ABB RobotStudio station: ProyectoC1.rspag

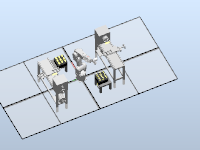
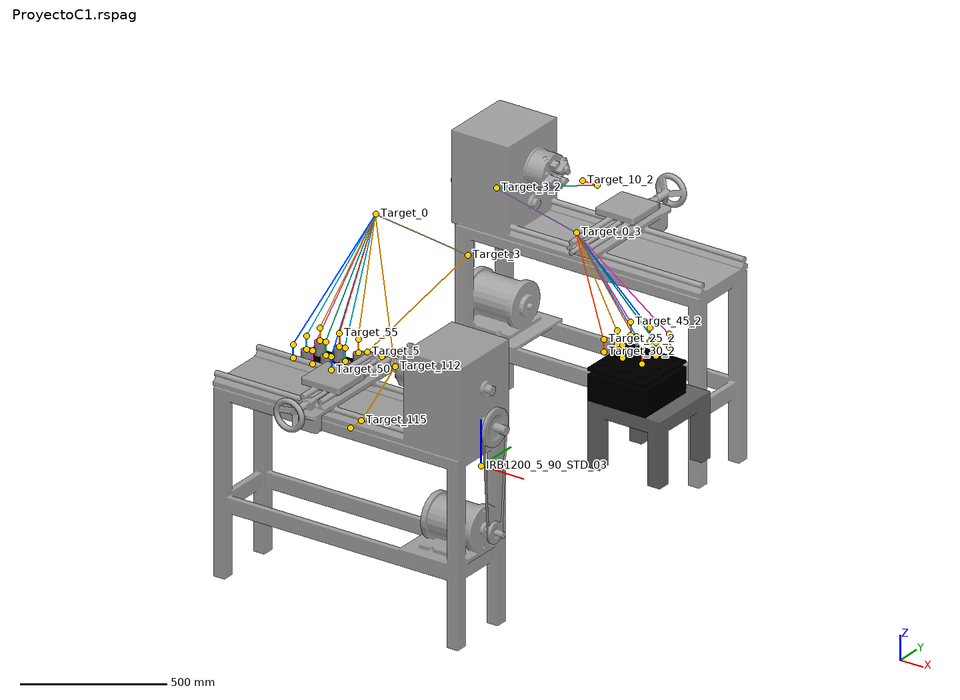
[picture v1: parts stored in the station drawn from their meshes, with robot base, taught points and paths (robot models come from the ABB library and are not in the file)]
--- station ---
Station Prueba1 (saved by RobotStudio 21.2.9526.0)
Controller Controller8
  mechanical unit ROB_1: IRB1200_5_90_STD_03, 6 joints, base frame (0, 0, 0) mm, rotated rx 0 ry 0 rz 180 deg
Layout (positions relative to the parent item):
  - Part_10 [part] at (300, 200, 0) mm, size 304.8 x 304.8 x 257.1 mm
  - IRB1200_5_90_STD_03 [mechanism, from Robots\IRB1200_5_90_STD_03.rslib] at (0, 0, 0) mm, rotated rx 0 ry 0 rz 180 deg; joint values [0.2272, -0.2553, -0.0183, 1.0645, 1.1707, 0.1682] (rad or m)
  - Pieza mecanizada_2 [part] at (-340.99, -320.29, 378.02) mm, rotated rx 0.01 ry 0 rz -1.08 deg, size 40.5 x 40.5 x 50.8 mm
  - Pieza mecanizada_3 [part] at (-340.26, -399.91, 378.02) mm, rotated rx 0 ry 0 rz 0.16 deg, size 40.5 x 40.5 x 50.8 mm
  - Pieza mecanizada_4 [part] at (-420.52, -241.71, 378.02) mm, rotated rx 0 ry 0 rz 2.15 deg, size 40.5 x 40.5 x 50.8 mm
  - Pieza mecanizada_5 [part] at (-420.06, -320.35, 378.02) mm, rotated rx 0 ry 0 rz 0.63 deg, size 40.5 x 40.5 x 50.8 mm
  - Pieza mecanizada_6 [part] at (-419.99, -400.08, 378.02) mm, size 40.5 x 40.5 x 50.8 mm
  - Pieza mecanizada_7 [part] at (-500.46, -240.05, 378.02) mm, rotated rx 0 ry 0 rz 0.98 deg, size 40.5 x 40.5 x 50.8 mm
  - Pieza mecanizada_8 [part] at (-500, -320, 378.02) mm, rotated rx 0 ry 0 rz 0.01 deg, size 40.5 x 40.5 x 50.8 mm
  - Pieza mecanizada_9 [part] at (-500, -400, 378.02) mm, rotated rx 0 ry 0 rz 0.01 deg, size 40.5 x 40.5 x 50.8 mm
  - Gripper_triple [mechanism] at (-326.49, -143.26, 968.24) mm, rotated rx 109.8 ry 16.48 rz -12.76 deg
      TCP Tool_acople at (0, -72.83, 94.3) mm, rotated rx 45 ry 0 rz 0 deg
      TCP Tool_desacople at (-1.73, 75.04, 92.27) mm, rotated rx -45 ry 0 rz 0 deg
      TCP Refrigerator at (40, 0, 44) mm, rotated rx 0 ry 90 rz 0 deg
      links: Herramienta
  - Torno_1 [smart component]
      signals: DO Finish, DO Mounted, DI Start, DI Attach, DI Detach
      connections:
        Torno_1.Start -> Timer_2.Active
        Timer_2.Output -> Torno_1.Finish
        Torno_1.Start -> LogicGate.InputA
        LogicGate.Output -> Detacher_10.Execute
        LineSensor.SensorOut -> Torno_1.Mounted
        Torno_1.Start -> Attacher.Execute
        LogicGate.Output -> Attacher_12.Execute
        Torno_1.Start -> Detacher_12.Execute
        LineSensor.SensedPart => Attacher.Child
        LineSensor.SensedPart => Detacher_10.Child
        LineSensor.SensedPart => Attacher_12.Child
        LineSensor.SensedPart => Detacher_12.Child
    - Torno [part] at (-288, 524, 0) mm, size 1289.1 x 1431.5 x 1343.8 mm
    - Detacher_10 [smart component, from Components\Detacher.rslib]
        properties: Child=Pieza mecanizada; KeepPosition=true
    - Attacher [smart component, from Components\Attacher.rslib]
        properties: Parent=Torno; Flange=0; Child=Pieza mecanizada; Mount=false; Offset=[0 0 0]; Orientation=[0 0 0]
    - LogicGate [smart component, from Components\LogicGate.rslib]
        properties: Operator=NOT; Delay=0
    - LineSensor [smart component, from Components\LineSensor.rslib]
        properties: Start=[0.14 -0.8 0.75]; End=[0.14 -0.69 0.75]; Radius=0; SensedPart=Pieza mecanizada; SensedPoint=[0.14 -0.777924682617188 0.75]
      - _sensorPart_ [part], size 0 x 110 x 0 mm
    - Attacher_12 [smart component, from Components\Attacher.rslib]
        properties: Parent=Gripper_triple; Flange=1; Child=Pieza mecanizada; Mount=false; Offset=[0 0 0]; Orientation=[0 0 0]
    - Detacher_12 [smart component, from Components\Detacher.rslib]
        properties: Child=Pieza mecanizada; KeepPosition=true
    - Torno_abierto [part] at (726.53, 140.46, 2.16) mm, size 1118.3 x 604.1 x 1068.7 mm
  - Torno_2 [smart component]
      signals: DO Finish, DO Mounted, DI Start, DI Attach, DI Detach
      connections:
        Torno_2.Start -> Attacher.Execute
        Torno_2.Start -> LogicGate_14.InputA
        LogicGate_14.Output -> Detacher.Execute
        LogicGate_14.Output -> Attacher_2.Execute
        Torno_2.Start -> Detacher_2.Execute
        LineSensor.SensorOut -> Torno_2.Mounted
        LineSensor.SensedPart => Detacher.Child
        LineSensor.SensedPart => Detacher_2.Child
        LineSensor.SensedPart => Attacher_2.Child
        LineSensor.SensedPart => Attacher.Child
    - Torno_3 [part] at (288, -524, 0) mm, rotated rx 0 ry 0 rz 180 deg, size 1289.1 x 1431.5 x 1343.8 mm
    - Attacher [smart component, from Components\Attacher.rslib]
        properties: Parent=Torno_3; Flange=0; Child=(none); Mount=false; Offset=[0 0 0]; Orientation=[0 0 0]
    - Attacher_2 [smart component, from Components\Attacher.rslib]
        properties: Parent=Gripper_triple; Flange=1; Child=(none); Mount=false; Offset=[0 0 0]; Orientation=[0 0 0]
    - Detacher [smart component, from Components\Detacher.rslib]
        properties: Child=(none); KeepPosition=true
    - Detacher_2 [smart component, from Components\Detacher.rslib]
        properties: Child=(none); KeepPosition=true
    - LineSensor [smart component, from Components\LineSensor.rslib]
        properties: Start=[-0.14 0.8 0.75]; End=[-0.14 0.69 0.75]; Radius=0; SensedPart=(none); SensedPoint=[0 0 0]
      - _sensorPart_ [part], size 0 x 110 x 0 mm
    - LogicGate_14 [smart component, from Components\LogicGate.rslib]
        properties: Operator=NOT; Delay=0
    - Torno_abierto_2 [part] at (-725.71, -155.46, 2.16) mm, rotated rx 0 ry 0 rz 180 deg, size 1118.3 x 604.1 x 1068.7 mm
  - Rotador [smart component]
      signals: DI Start, DO Finish, DI Attach, DI Detach
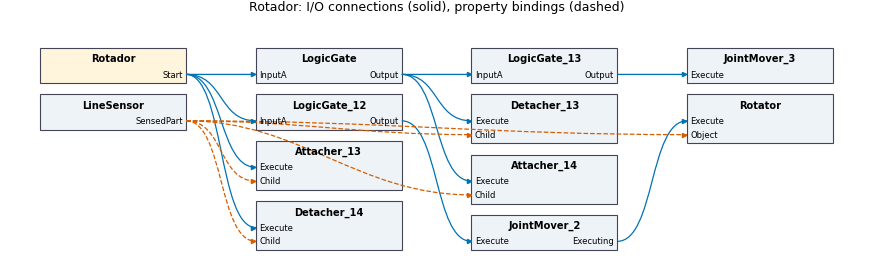
      connections:
        Rotador.Start -> LogicGate.InputA
        Rotador.Start -> Attacher_13.Execute
        LogicGate.Output -> Detacher_13.Execute
        Rotador.Start -> LogicGate_12.InputA
        LogicGate_12.Output -> JointMover_2.Execute
        LogicGate.Output -> Attacher_14.Execute
        Rotador.Start -> Detacher_14.Execute
        JointMover_2.Executing -> Rotator.Execute
        LogicGate.Output -> LogicGate_13.InputA
        LogicGate_13.Output -> JointMover_3.Execute
        LineSensor.SensedPart => Attacher_13.Child
        LineSensor.SensedPart => Detacher_13.Child
        LineSensor.SensedPart => Detacher_14.Child
        LineSensor.SensedPart => Attacher_14.Child
        LineSensor.SensedPart => Rotator.Object
    - My_Mechanism [mechanism] at (0, 0, 0) mm; joint values [0] (rad or m)
        links: L0, L1
    - JointMover_2 [smart component, from Components\JointMover.rslib]
        properties: Mechanism=My_Mechanism; Relative=false; Duration=0.5; J1=3.14159265358979
    - JointMover_3 [smart component, from Components\JointMover.rslib]
        properties: Mechanism=My_Mechanism; Relative=false; Duration=1; J1=0
    - LogicGate [smart component, from Components\LogicGate.rslib]
        properties: Operator=NOT; Delay=0
    - Attacher_13 [smart component, from Components\Attacher.rslib]
        properties: Parent=My_Mechanism; Flange=0; Child=(none); Mount=false; Offset=[0 0 0]; Orientation=[0 0 0]
    - LineSensor [smart component, from Components\LineSensor.rslib]
        properties: Start=[-0.42 -0.225 0.16]; End=[-0.42 -0.225 0.06]; Radius=0; SensedPart=(none); SensedPoint=[0 0 0]
      - _sensorPart_ [part], size 0 x 0 x 100 mm
    - Detacher_13 [smart component, from Components\Detacher.rslib]
        properties: Child=(none); KeepPosition=true
    - LogicGate_12 [smart component, from Components\LogicGate.rslib]
        properties: Operator=OR; Delay=2
    - Attacher_14 [smart component, from Components\Attacher.rslib]
        properties: Parent=Gripper_triple; Flange=0; Child=(none); Mount=false; Offset=[0 0 0]; Orientation=[0 0 0]
    - Detacher_14 [smart component, from Components\Detacher.rslib]
        properties: Child=(none); KeepPosition=true
    - Rotator [smart component, from Components\Rotator.rslib]
        properties: Object=(none); CenterPoint=[-0.54 -0.225 0.108]; Axis=[1 0 0]; Speed=11.8682389135614; Reference=Global; ReferenceObject=(none)
    - Timer [smart component, from Components\Timer.rslib]
        properties: StartTime=0; Interval=0; Repeat=true; CurrentTime=1.512
    - LogicGate_13 [smart component, from Components\LogicGate.rslib]
        properties: Operator=OR; Delay=2
  - Sensor_sin_maquinar [smart component]
      signals: DO Sensor_1_activo, DO Sensor_2_activo, DO Sensor_3_activo, DO Sensor_4_activo, DO Sensor_5_activo, DO Sensor_6_activo, DO Sensor_7_activo, DO Sensor_8_activo, DO Sensor_9_activo
      connections:
        LineSensor_4.SensorOut -> Sensor_sin_maquinar.Sensor_4_activo
        LineSensor_5.SensorOut -> Sensor_sin_maquinar.Sensor_5_activo
        LineSensor_6.SensorOut -> Sensor_sin_maquinar.Sensor_6_activo
        LineSensor_7.SensorOut -> Sensor_sin_maquinar.Sensor_7_activo
        LineSensor_8.SensorOut -> Sensor_sin_maquinar.Sensor_8_activo
        LineSensor_9.SensorOut -> Sensor_sin_maquinar.Sensor_9_activo
        LineSensor.SensorOut -> Sensor_sin_maquinar.Sensor_1_activo
        LineSensor_2.SensorOut -> Sensor_sin_maquinar.Sensor_2_activo
        LineSensor_3.SensorOut -> Sensor_sin_maquinar.Sensor_3_activo
    - Palet_2 [part] at (-300, -200, 250) mm, rotated rx 0 ry 0 rz 180 deg, size 243.8 x 243.8 x 129.5 mm
    - LineSensor [smart component, from Components\LineSensor.rslib]
        properties: Start=[-0.37 -0.240108 0.4]; End=[-0.31 -0.24 0.4]; Radius=0; SensedPart=(none); SensedPoint=[0 0 0]
      - _sensorPart_ [part], size 60 x 0.1 x 0 mm
    - LineSensor_2 [smart component, from Components\LineSensor.rslib]
        properties: Start=[-0.37 -0.32 0.4]; End=[-0.31 -0.32 0.4]; Radius=0; SensedPart=Pieza mecanizada_2; SensedPoint=[-0.361003173828125 -0.32 0.4]
      - _sensorPart_ [part], size 60 x 0 x 0 mm
    - LineSensor_3 [smart component, from Components\LineSensor.rslib]
        properties: Start=[-0.37 -0.4 0.4]; End=[-0.31 -0.4 0.4]; Radius=0; SensedPart=Pieza mecanizada_3; SensedPoint=[-0.360261657714844 -0.4 0.4]
      - _sensorPart_ [part], size 60 x 0 x 0 mm
    - LineSensor_4 [smart component, from Components\LineSensor.rslib]
        properties: Start=[-0.45 -0.24 0.4]; End=[-0.39 -0.24 0.4]; Radius=0; SensedPart=Pieza mecanizada_4; SensedPoint=[-0.440390747070313 -0.24 0.4]
      - _sensorPart_ [part], size 60 x 0 x 0 mm
    - LineSensor_5 [smart component, from Components\LineSensor.rslib]
        properties: Start=[-0.45 -0.32 0.4]; End=[-0.39 -0.32 0.4]; Radius=0; SensedPart=Pieza mecanizada_5; SensedPoint=[-0.440016571044922 -0.319999969482422 0.4]
      - _sensorPart_ [part], size 60 x 0 x 0 mm
    - LineSensor_6 [smart component, from Components\LineSensor.rslib]
        properties: Start=[-0.45 -0.4 0.4]; End=[-0.39 -0.4 0.4]; Radius=0; SensedPart=Pieza mecanizada_6; SensedPoint=[-0.439984832763672 -0.4 0.4]
      - _sensorPart_ [part], size 60 x 0 x 0 mm
    - LineSensor_7 [smart component, from Components\LineSensor.rslib]
        properties: Start=[-0.53 -0.24 0.4]; End=[-0.47 -0.24 0.4]; Radius=0; SensedPart=Pieza mecanizada_7; SensedPoint=[-0.520428344726563 -0.239999984741211 0.4]
      - _sensorPart_ [part], size 60 x 0 x 0 mm
    - LineSensor_8 [smart component, from Components\LineSensor.rslib]
        properties: Start=[-0.53 -0.32 0.4]; End=[-0.47 -0.32 0.4]; Radius=0; SensedPart=Pieza mecanizada_8; SensedPoint=[-0.520002136230469 -0.319999969482422 0.4]
      - _sensorPart_ [part], size 60 x 0 x 0 mm
    - LineSensor_9 [smart component, from Components\LineSensor.rslib]
        properties: Start=[-0.53 -0.4 0.4]; End=[-0.47 -0.4 0.4]; Radius=0; SensedPart=Pieza mecanizada_9; SensedPoint=[-0.520002685546875 -0.399999969482422 0.4]
      - _sensorPart_ [part], size 60 x 0 x 0 mm
  - Sensor_maquinadas [smart component]
      signals: DO Sensor_1_activo, DO Sensor_2_activo, DO Sensor_3_activo, DO Sensor_4_activo, DO Sensor_5_activo, DO Sensor_6_activo, DO Sensor_7_activo, DO Sensor_8_activo, DO Sensor_9_activo, DI Detach
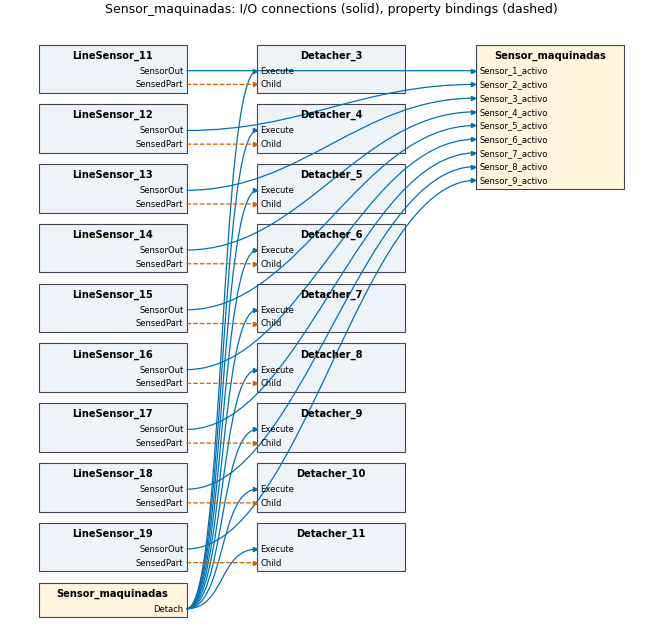
      connections:
        LineSensor_11.SensorOut -> Sensor_maquinadas.Sensor_1_activo
        LineSensor_12.SensorOut -> Sensor_maquinadas.Sensor_2_activo
        LineSensor_13.SensorOut -> Sensor_maquinadas.Sensor_3_activo
        LineSensor_14.SensorOut -> Sensor_maquinadas.Sensor_4_activo
        LineSensor_15.SensorOut -> Sensor_maquinadas.Sensor_5_activo
        LineSensor_16.SensorOut -> Sensor_maquinadas.Sensor_6_activo
        LineSensor_17.SensorOut -> Sensor_maquinadas.Sensor_7_activo
        LineSensor_18.SensorOut -> Sensor_maquinadas.Sensor_8_activo
        LineSensor_19.SensorOut -> Sensor_maquinadas.Sensor_9_activo
        Sensor_maquinadas.Detach -> Detacher_3.Execute
        Sensor_maquinadas.Detach -> Detacher_4.Execute
        Sensor_maquinadas.Detach -> Detacher_5.Execute
        Sensor_maquinadas.Detach -> Detacher_6.Execute
        Sensor_maquinadas.Detach -> Detacher_7.Execute
        Sensor_maquinadas.Detach -> Detacher_8.Execute
        Sensor_maquinadas.Detach -> Detacher_9.Execute
        Sensor_maquinadas.Detach -> Detacher_10.Execute
        Sensor_maquinadas.Detach -> Detacher_11.Execute
        LineSensor_11.SensedPart => Detacher_3.Child
        LineSensor_12.SensedPart => Detacher_4.Child
        LineSensor_13.SensedPart => Detacher_5.Child
        LineSensor_14.SensedPart => Detacher_6.Child
        LineSensor_15.SensedPart => Detacher_7.Child
        LineSensor_16.SensedPart => Detacher_8.Child
        LineSensor_17.SensedPart => Detacher_9.Child
        LineSensor_18.SensedPart => Detacher_10.Child
        LineSensor_19.SensedPart => Detacher_11.Child
    - Palet [part] at (300, 200, 250) mm, size 242.1 x 242.1 x 126.4 mm
    - LineSensor_11 [smart component, from Components\LineSensor.rslib]
        properties: Start=[0.37 0.240108 0.4]; End=[0.31 0.24 0.4]; Radius=0; SensedPart=(none); SensedPoint=[0 0 0]
      - _sensorPart_ [part], size 60 x 0.1 x 0 mm
    - LineSensor_12 [smart component, from Components\LineSensor.rslib]
        properties: Start=[0.37 0.32 0.4]; End=[0.31 0.32 0.4]; Radius=0; SensedPart=Palet; SensedPoint=[0.360499572753906 0.32 0.375]
      - _sensorPart_ [part], size 60 x 0 x 0 mm
    - LineSensor_13 [smart component, from Components\LineSensor.rslib]
        properties: Start=[0.37 0.4 0.4]; End=[0.31 0.4 0.4]; Radius=0; SensedPart=Palet; SensedPoint=[0.360499572753906 0.4 0.375]
      - _sensorPart_ [part], size 60 x 0 x 0 mm
    - LineSensor_14 [smart component, from Components\LineSensor.rslib]
        properties: Start=[0.45 0.24 0.4]; End=[0.39 0.24 0.4]; Radius=0; SensedPart=(none); SensedPoint=[0 0 0]
      - _sensorPart_ [part], size 60 x 0 x 0 mm
    - LineSensor_15 [smart component, from Components\LineSensor.rslib]
        properties: Start=[0.45 0.32 0.4]; End=[0.39 0.32 0.4]; Radius=0; SensedPart=(none); SensedPoint=[0 0 0]
      - _sensorPart_ [part], size 60 x 0 x 0 mm
    - LineSensor_16 [smart component, from Components\LineSensor.rslib]
        properties: Start=[0.45 0.4 0.4]; End=[0.39 0.4 0.4]; Radius=0; SensedPart=(none); SensedPoint=[0 0 0]
      - _sensorPart_ [part], size 60 x 0 x 0 mm
    - LineSensor_17 [smart component, from Components\LineSensor.rslib]
        properties: Start=[0.53 0.24 0.4]; End=[0.47 0.24 0.4]; Radius=0; SensedPart=(none); SensedPoint=[0 0 0]
      - _sensorPart_ [part], size 60 x 0 x 0 mm
    - LineSensor_18 [smart component, from Components\LineSensor.rslib]
        properties: Start=[0.53 0.32 0.4]; End=[0.47 0.32 0.4]; Radius=0; SensedPart=(none); SensedPoint=[0 0 0]
      - _sensorPart_ [part], size 60 x 0 x 0 mm
    - LineSensor_19 [smart component, from Components\LineSensor.rslib]
        properties: Start=[0.53 0.4 0.4]; End=[0.47 0.4 0.4]; Radius=0; SensedPart=(none); SensedPoint=[0 0 0]
      - _sensorPart_ [part], size 60 x 0 x 0 mm
    - Detacher_3 [smart component, from Components\Detacher.rslib]
        properties: Child=(none); KeepPosition=true
    - Detacher_4 [smart component, from Components\Detacher.rslib]
        properties: Child=Palet; KeepPosition=true
    - Detacher_5 [smart component, from Components\Detacher.rslib]
        properties: Child=Palet; KeepPosition=true
    - Detacher_6 [smart component, from Components\Detacher.rslib]
        properties: Child=(none); KeepPosition=true
    - Detacher_7 [smart component, from Components\Detacher.rslib]
        properties: Child=(none); KeepPosition=true
    - Detacher_8 [smart component, from Components\Detacher.rslib]
        properties: Child=(none); KeepPosition=true
    - Detacher_9 [smart component, from Components\Detacher.rslib]
        properties: Child=(none); KeepPosition=true
    - Detacher_10 [smart component, from Components\Detacher.rslib]
        properties: Child=(none); KeepPosition=true
    - Detacher_11 [smart component, from Components\Detacher.rslib]
        properties: Child=(none); KeepPosition=true
  - Attacher [smart component, from Components\Attacher.rslib]
      properties: Parent=Gripper_triple; Flange=0; Child=Pieza mecanizada; Mount=false; Offset=[0 0 0]; Orientation=[0 0 0]
  - Attacher_2 [smart component, from Components\Attacher.rslib]
      properties: Parent=Gripper_triple; Flange=0; Child=Pieza mecanizada_2; Mount=false; Offset=[0 0 0]; Orientation=[0 0 0]
  - Attacher_3 [smart component, from Components\Attacher.rslib]
      properties: Parent=Gripper_triple; Flange=0; Child=Pieza mecanizada_3; Mount=false; Offset=[0 0 0]; Orientation=[0 0 0]
  - Attacher_4 [smart component, from Components\Attacher.rslib]
      properties: Parent=Gripper_triple; Flange=0; Child=Pieza mecanizada_4; Mount=false; Offset=[0 0 0]; Orientation=[0 0 0]
  - Attacher_5 [smart component, from Components\Attacher.rslib]
      properties: Parent=Gripper_triple; Flange=0; Child=Pieza mecanizada_5; Mount=false; Offset=[0 0 0]; Orientation=[0 0 0]
  - Attacher_6 [smart component, from Components\Attacher.rslib]
      properties: Parent=Gripper_triple; Flange=0; Child=Pieza mecanizada_6; Mount=false; Offset=[0 0 0]; Orientation=[0 0 0]
  - Attacher_7 [smart component, from Components\Attacher.rslib]
      properties: Parent=Gripper_triple; Flange=0; Child=Pieza mecanizada_7; Mount=false; Offset=[0 0 0]; Orientation=[0 0 0]
  - Attacher_8 [smart component, from Components\Attacher.rslib]
      properties: Parent=Gripper_triple; Flange=0; Child=Pieza mecanizada_8; Mount=false; Offset=[0 0 0]; Orientation=[0 0 0]
  - Attacher_9 [smart component, from Components\Attacher.rslib]
      properties: Parent=Gripper_triple; Flange=0; Child=Pieza mecanizada_9; Mount=false; Offset=[0 0 0]; Orientation=[0 0 0]
  - Attacher_10 [smart component, from Components\Attacher.rslib]
      properties: Parent=Gripper_triple; Flange=0; Child=(none); Mount=false; Offset=[0 0 0]; Orientation=[0 0 0]
  - LogicGate_2 [smart component, from Components\LogicGate.rslib]
      properties: Operator=AND; Delay=0
  - LogicGate_3 [smart component, from Components\LogicGate.rslib]
      properties: Operator=AND; Delay=0
  - LogicGate_4 [smart component, from Components\LogicGate.rslib]
      properties: Operator=AND; Delay=0
  - LogicGate_5 [smart component, from Components\LogicGate.rslib]
      properties: Operator=AND; Delay=0
  - LogicGate_6 [smart component, from Components\LogicGate.rslib]
      properties: Operator=AND; Delay=0
  - LogicGate_7 [smart component, from Components\LogicGate.rslib]
      properties: Operator=AND; Delay=0
  - LogicGate_8 [smart component, from Components\LogicGate.rslib]
      properties: Operator=AND; Delay=0
  - LogicGate_9 [smart component, from Components\LogicGate.rslib]
      properties: Operator=AND; Delay=0
  - LogicGate_10 [smart component, from Components\LogicGate.rslib]
      properties: Operator=AND; Delay=0
  - Pieza mecanizada [part] at (-339.54, -240.41, 378.02) mm, rotated rx 0 ry 0 rz -1.05 deg, size 40.5 x 40.5 x 50.8 mm
  - Detacher [smart component, from Components\Detacher.rslib]
      properties: Child=Pieza mecanizada; KeepPosition=true
  - Detacher_2 [smart component, from Components\Detacher.rslib]
      properties: Child=Pieza mecanizada_2; KeepPosition=true
  - Detacher_3 [smart component, from Components\Detacher.rslib]
      properties: Child=Pieza mecanizada_3; KeepPosition=true
  - Detacher_4 [smart component, from Components\Detacher.rslib]
      properties: Child=Pieza mecanizada_4; KeepPosition=true
  - Detacher_5 [smart component, from Components\Detacher.rslib]
      properties: Child=Pieza mecanizada_5; KeepPosition=true
  - Detacher_6 [smart component, from Components\Detacher.rslib]
      properties: Child=Pieza mecanizada_6; KeepPosition=true
  - Detacher_7 [smart component, from Components\Detacher.rslib]
      properties: Child=Pieza mecanizada_7; KeepPosition=true
  - Detacher_8 [smart component, from Components\Detacher.rslib]
      properties: Child=Pieza mecanizada_8; KeepPosition=true
  - Detacher_9 [smart component, from Components\Detacher.rslib]
      properties: Child=Pieza mecanizada_9; KeepPosition=true
  - LogicGate_11 [smart component, from Components\LogicGate.rslib]
      properties: Operator=AND; Delay=0
Attachment: Gripper_triple is attached to IRB1200_5_90_STD_03 / Link6
Station signals: DI Execute
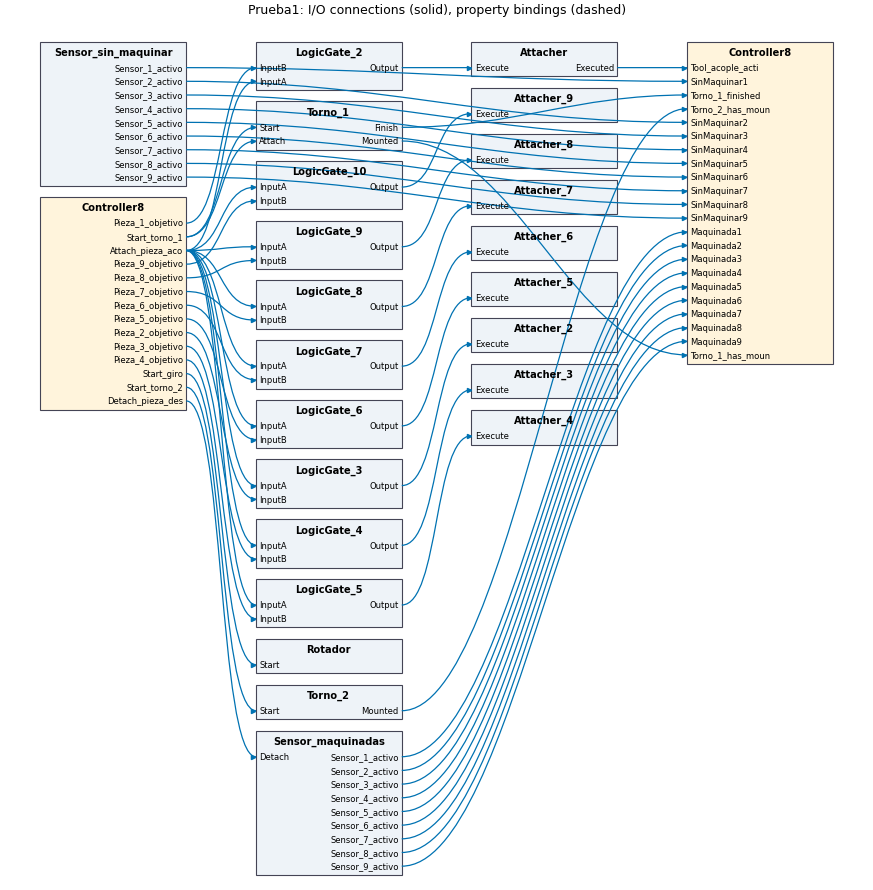
Station logic (signal -> signal, property => property):
  Attacher.Executed -> Controller8.Tool_acople_activa
  Sensor_sin_maquinar.Sensor_1_activo -> Controller8.SinMaquinar1
  Controller8.Pieza_1_objetivo -> LogicGate_2.InputB
  LogicGate_2.Output -> Attacher.Execute
  Controller8.Start_torno_1 -> Torno_1.Start
  Torno_1.Finish -> Controller8.Torno_1_finished
  Controller8.Attach_pieza_acople -> LogicGate_3.InputA
  Controller8.Attach_pieza_acople -> LogicGate_4.InputA
  Controller8.Attach_pieza_acople -> LogicGate_5.InputA
  Controller8.Attach_pieza_acople -> LogicGate_2.InputA
  Controller8.Attach_pieza_acople -> LogicGate_6.InputA
  Controller8.Attach_pieza_acople -> LogicGate_7.InputA
  Controller8.Attach_pieza_acople -> LogicGate_8.InputA
  Controller8.Attach_pieza_acople -> LogicGate_9.InputA
  Controller8.Attach_pieza_acople -> LogicGate_10.InputA
  Controller8.Pieza_9_objetivo -> LogicGate_10.InputB
  Controller8.Pieza_8_objetivo -> LogicGate_9.InputB
  Controller8.Pieza_7_objetivo -> LogicGate_8.InputB
  Controller8.Pieza_6_objetivo -> LogicGate_7.InputB
  Controller8.Pieza_5_objetivo -> LogicGate_6.InputB
  Controller8.Pieza_2_objetivo -> LogicGate_3.InputB
  Controller8.Pieza_3_objetivo -> LogicGate_4.InputB
  Controller8.Pieza_4_objetivo -> LogicGate_5.InputB
  Controller8.Start_torno_1 -> Torno_1.Attach
  Torno_2.Mounted -> Controller8.Torno_2_has_mounted
  Sensor_sin_maquinar.Sensor_2_activo -> Controller8.SinMaquinar2
  Sensor_sin_maquinar.Sensor_3_activo -> Controller8.SinMaquinar3
  Sensor_sin_maquinar.Sensor_4_activo -> Controller8.SinMaquinar4
  Sensor_sin_maquinar.Sensor_5_activo -> Controller8.SinMaquinar5
  Sensor_sin_maquinar.Sensor_6_activo -> Controller8.SinMaquinar6
  Sensor_sin_maquinar.Sensor_7_activo -> Controller8.SinMaquinar7
  Sensor_sin_maquinar.Sensor_8_activo -> Controller8.SinMaquinar8
  Sensor_sin_maquinar.Sensor_9_activo -> Controller8.SinMaquinar9
  LogicGate_3.Output -> Attacher_2.Execute
  LogicGate_4.Output -> Attacher_3.Execute
  LogicGate_5.Output -> Attacher_4.Execute
  LogicGate_6.Output -> Attacher_5.Execute
  LogicGate_7.Output -> Attacher_6.Execute
  LogicGate_8.Output -> Attacher_7.Execute
  LogicGate_9.Output -> Attacher_8.Execute
  LogicGate_10.Output -> Attacher_9.Execute
  Controller8.Start_giro -> Rotador.Start
  Controller8.Start_torno_2 -> Torno_2.Start
  Controller8.Detach_pieza_desacople -> Sensor_maquinadas.Detach
  Sensor_maquinadas.Sensor_1_activo -> Controller8.Maquinada1
  Sensor_maquinadas.Sensor_2_activo -> Controller8.Maquinada2
  Sensor_maquinadas.Sensor_3_activo -> Controller8.Maquinada3
  Sensor_maquinadas.Sensor_4_activo -> Controller8.Maquinada4
  Sensor_maquinadas.Sensor_5_activo -> Controller8.Maquinada5
  Sensor_maquinadas.Sensor_6_activo -> Controller8.Maquinada6
  Sensor_maquinadas.Sensor_7_activo -> Controller8.Maquinada7
  Sensor_maquinadas.Sensor_8_activo -> Controller8.Maquinada8
  Sensor_maquinadas.Sensor_9_activo -> Controller8.Maquinada9
  Torno_1.Mounted -> Controller8.Torno_1_has_mounted
Targets, tools, work objects and paths stored in the station and not in the controller backup, written as RAPID:
! task T_ROB1
MODULE Module1
  CONST robtarget Target_20:=[[11.107639525,-224.886782499,425.07180983],[0.006192071,-0.700860473,0.006192057,-0.713244638],[0,1,0,0],[9E+09,9E+09,9E+09,9E+09,9E+09,9E+09]];
  CONST robtarget Target_0_2:=[[-390.352989081,345.323504999,617.602499755],[0.036729233,-0.769016339,0.224591957,-0.597346873],[0,0,-2,7],[9E+09,9E+09,9E+09,9E+09,9E+09,9E+09]];
  CONST robtarget Target_1_2:=[[10.580526231,345.323509175,617.602503568],[0.396416501,0.702587169,0.384966146,0.44835956],[-2,0,-1,2],[9E+09,9E+09,9E+09,9E+09,9E+09,9E+09]];
  CONST robtarget Target_2_2:=[[30.118499272,290.328983403,602.616663519],[0.258418789,0.681263439,-0.456625437,0.51048317],[1,-1,0,0],[9E+09,9E+09,9E+09,9E+09,9E+09,9E+09]];
  CONST robtarget Target_20_2:=[[11.107639525,-224.886782499,425.07180983],[0.006192071,-0.700860473,0.006192057,-0.713244638],[0,1,0,0],[9E+09,9E+09,9E+09,9E+09,9E+09,9E+09]];
ENDMODULE


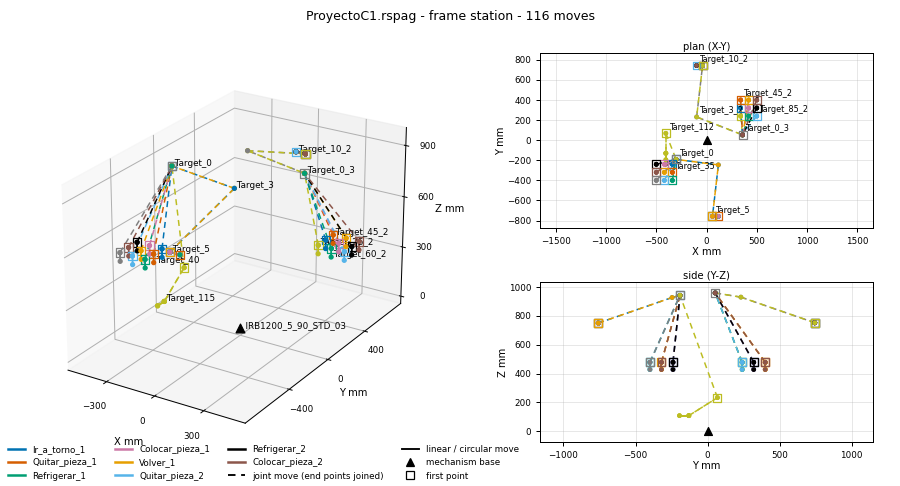
[picture p0: tool path of ProyectoC1.rspag in frame station, 116 of 116 moves have a stored position in this frame; points joined in program order, loops and branches not executed]
--- Backups/Controller8/RAPID/TASK1/PROGMOD/CalibData.mod ---
MODULE CalibData
    PERS tooldata Tool_acople:=[TRUE,[[0,-72.833,94.303],[0.92388,0.382683,0,0]],[1.818,[0,0,57],[1,0,0,0],0,0,0]];
    PERS tooldata Tool_desacople:=[TRUE,[[-1.732,75.041,92.274],[0,0,0.382683,0.92388]],[1.818,[0,0,57],[1,0,0,0],0,0,0]];
    PERS tooldata Refrigerator:=[TRUE,[[40,0,44],[0.5,0.5,0.5,0.5]],[1.818,[0,0,57],[1,0,0,0],0,0,0]];
    TASK PERS wobjdata Workobject_1:=[FALSE,TRUE,"",[[-300,-200,250],[1,0,0,0]],[[0,0,125],[1,0,0,0]]];
    TASK PERS wobjdata Workobject_2:=[FALSE,TRUE,"",[[300,200,250],[0,0,0,1]],[[0,0,125],[1,0,0,0]]];
    TASK PERS wobjdata Workobject_3:=[FALSE,TRUE,"",[[88,-536.5,325],[1,0,0,0]],[[0,0,0],[1,0,0,0]]];
    TASK PERS wobjdata Workobject_4:=[FALSE,TRUE,"",[[-68,521.5,327.5],[0,0,0,1]],[[0,0,0],[1,0,0,0]]];
ENDMODULE

--- Backups/Controller8/RAPID/TASK1/PROGMOD/Module1.mod ---
MODULE Module1
        CONST robtarget Target_5:=[[-28.75,-221.875,425],[0,0.707106781,0,0.707106781],[0,1,-2,0],[9E+09,9E+09,9E+09,9E+09,9E+09,9E+09]];
    CONST robtarget Target_10:=[[31.25,-221.875,425],[0,0.707106781,0,0.707106781],[0,1,-2,0],[9E+09,9E+09,9E+09,9E+09,9E+09,9E+09]];
    CONST robtarget Target_0:=[[-390.352989081,345.323504999,617.602499755],[0.036729233,-0.769016339,0.224591957,-0.597346873],[0,1,-1,0],[9E+09,9E+09,9E+09,9E+09,9E+09,9E+09]];
    CONST robtarget Target_1:=[[10.580526231,345.323509175,617.602503568],[0.396416501,0.702587169,0.384966146,0.44835956],[1,-1,1,0],[9E+09,9E+09,9E+09,9E+09,9E+09,9E+09]];
    CONST robtarget Target_2:=[[30.118499272,290.328983403,602.616663519],[0.258418789,0.681263439,-0.456625437,0.51048317],[1,-1,0,0],[9E+09,9E+09,9E+09,9E+09,9E+09,9E+09]];
    CONST robtarget Target_3:=[[30.118503807,290.32899798,602.616712274],[0.034631434,-0.818597309,0.050250854,-0.571116417],[0,0,-1,0],[9E+09,9E+09,9E+09,9E+09,9E+09,9E+09]];
    CONST robtarget Target_6:=[[11.25,-251.875,425],[0,0.707106781,0,0.707106781],[1,0,0,1],[9E+09,9E+09,9E+09,9E+09,9E+09,9E+09]];
    CONST robtarget Target_7:=[[11.25,-191.875,425],[0,0.707106781,0,0.707106781],[1,0,0,1],[9E+09,9E+09,9E+09,9E+09,9E+09,9E+09]];
    CONST robtarget Target_10_2:=[[31.25,-221.875,425],[0,0.707106781,0,0.707106781],[-2,1,-2,0],[9E+09,9E+09,9E+09,9E+09,9E+09,9E+09]];
    CONST robtarget Target_5_2:=[[-28.75,-221.875,425],[0,0.707106781,0,0.707106781],[-2,1,-2,0],[9E+09,9E+09,9E+09,9E+09,9E+09,9E+09]];
    CONST robtarget Target_3_2:=[[30.118503807,290.32899798,602.616712274],[0.034631434,-0.818597309,0.050250854,-0.571116417],[-2,0,-1,0],[9E+09,9E+09,9E+09,9E+09,9E+09,9E+09]];
!***********************************************************
    !
    ! Module:  Module1
    !
    ! Description:
    !   <Insert description here>
    !
    ! Author: ManuelEsteban
    !
    ! Version: 1.0
    !
    !***********************************************************


    !***********************************************************
    !
    ! Procedure main
    !
    !   This is the entry point of your program
    !
    !***********************************************************
    VAR num contador_sin_maquinar:=0;
    VAR num contador_maquinadas:=0;
    VAR bool continue := TRUE;
    CONST robtarget Target_25:=[[-39.985,-40.086,103.016],[0,-0.707106781,0.707106781,0],[0,1,-1,1],[9E+09,9E+09,9E+09,9E+09,9E+09,9E+09]];
    CONST robtarget Target_30:=[[-39.985,-40.086,53.016],[0,-0.707106781,0.707106781,0],[0,1,0,1],[9E+09,9E+09,9E+09,9E+09,9E+09,9E+09]];
    CONST robtarget Target_0_3:=[[-58.912153108,147.259134131,584.239861581],[0.653281498,-0.65328152,0.270598033,0.270597938],[-2,-1,-1,0],[9E+09,9E+09,9E+09,9E+09,9E+09,9E+09]];
    CONST robtarget Target_35:=[[-39.956,-119.973,103.016],[0,-0.707106781,0.707106781,0],[0,1,-1,1],[9E+09,9E+09,9E+09,9E+09,9E+09,9E+09]];
    CONST robtarget Target_40:=[[-39.956,-119.973,53.016],[0,-0.707106781,0.707106781,0],[0,1,0,1],[9E+09,9E+09,9E+09,9E+09,9E+09,9E+09]];
    CONST robtarget Target_45:=[[-39.99,-200.054,103.016],[0,-0.707106781,0.707106781,0],[0,1,0,1],[9E+09,9E+09,9E+09,9E+09,9E+09,9E+09]];
    CONST robtarget Target_50:=[[-39.99,-200.054,53.016],[0,-0.707106781,0.707106781,0],[0,1,0,1],[9E+09,9E+09,9E+09,9E+09,9E+09,9E+09]];
    CONST robtarget Target_55:=[[-119.955,-40.038,103.016],[0,-0.707106781,0.707106781,0],[0,1,-1,1],[9E+09,9E+09,9E+09,9E+09,9E+09,9E+09]];
    CONST robtarget Target_60:=[[-119.955,-40.038,53.016],[0,-0.707106781,0.707106781,0],[0,1,-1,1],[9E+09,9E+09,9E+09,9E+09,9E+09,9E+09]];
    CONST robtarget Target_65:=[[-119.958,-120.121,103.016],[0,-0.707106781,0.707106781,0],[0,1,-1,1],[9E+09,9E+09,9E+09,9E+09,9E+09,9E+09]];
    CONST robtarget Target_70:=[[-119.958,-120.121,53.016],[0,-0.707106781,0.707106781,0],[0,1,0,1],[9E+09,9E+09,9E+09,9E+09,9E+09,9E+09]];
    CONST robtarget Target_75:=[[-119.992,-200.079,103.016],[0,-0.707106781,0.707106781,0],[0,1,-1,1],[9E+09,9E+09,9E+09,9E+09,9E+09,9E+09]];
    CONST robtarget Target_80:=[[-119.992,-200.079,53.016],[0,-0.707106781,0.707106781,0],[0,1,0,1],[9E+09,9E+09,9E+09,9E+09,9E+09,9E+09]];
    CONST robtarget Target_85:=[[-200.003,-40.005,103.016],[0,-0.707106781,0.707106781,0],[0,1,-1,1],[9E+09,9E+09,9E+09,9E+09,9E+09,9E+09]];
    CONST robtarget Target_90:=[[-200.003,-40.005,53.016],[0,-0.707106781,0.707106781,0],[0,1,-1,1],[9E+09,9E+09,9E+09,9E+09,9E+09,9E+09]];
    CONST robtarget Target_95:=[[-200.003,-120.004,103.016],[0,-0.707106781,0.707106781,0],[0,1,-1,1],[9E+09,9E+09,9E+09,9E+09,9E+09,9E+09]];
    CONST robtarget Target_100:=[[-200.003,-120.004,53.016],[0,-0.707106781,0.707106781,0],[0,1,-1,1],[9E+09,9E+09,9E+09,9E+09,9E+09,9E+09]];
    CONST robtarget Target_105:=[[-200.003,-200.005,103.016],[0,-0.707106781,0.707106781,0],[0,1,-1,1],[9E+09,9E+09,9E+09,9E+09,9E+09,9E+09]];
    CONST robtarget Target_110:=[[-200.003,-200.005,53.016],[0,-0.707106781,0.707106781,0],[0,1,-1,1],[9E+09,9E+09,9E+09,9E+09,9E+09,9E+09]];
    CONST robtarget Target_0_4:=[[-390.352989081,345.323504999,617.602499755],[0.036729233,-0.769016339,0.224591957,-0.597346873],[0,1,-1,0],[9E+09,9E+09,9E+09,9E+09,9E+09,9E+09]];
    CONST robtarget Target_25_2:=[[-39.985,-40.086,103.016],[0,-0.707106781,0.707106781,0],[-2,-1,-1,0],[9E+09,9E+09,9E+09,9E+09,9E+09,9E+09]];
    CONST robtarget Target_30_2:=[[-39.985,-40.086,53.016],[0,-0.707106781,0.707106781,0],[-2,-1,0,0],[9E+09,9E+09,9E+09,9E+09,9E+09,9E+09]];
    CONST robtarget Target_35_2:=[[-39.956,-119.973,103.016],[0,-0.707106781,0.707106781,0],[-2,-1,-1,0],[9E+09,9E+09,9E+09,9E+09,9E+09,9E+09]];
    CONST robtarget Target_40_2:=[[-39.956,-119.973,53.016],[0,-0.707106781,0.707106781,0],[-2,-1,0,0],[9E+09,9E+09,9E+09,9E+09,9E+09,9E+09]];
    CONST robtarget Target_45_2:=[[-39.99,-200.054,103.016],[0,-0.707106781,0.707106781,0],[-2,-1,0,0],[9E+09,9E+09,9E+09,9E+09,9E+09,9E+09]];
    CONST robtarget Target_50_2:=[[-39.99,-200.054,53.016],[0,-0.707106781,0.707106781,0],[-2,-1,0,0],[9E+09,9E+09,9E+09,9E+09,9E+09,9E+09]];
    CONST robtarget Target_55_2:=[[-119.955,-40.038,103.016],[0,-0.707106781,0.707106781,0],[-2,-1,-1,0],[9E+09,9E+09,9E+09,9E+09,9E+09,9E+09]];
    CONST robtarget Target_60_2:=[[-119.955,-40.038,53.016],[0,-0.707106781,0.707106781,0],[-2,-1,-1,0],[9E+09,9E+09,9E+09,9E+09,9E+09,9E+09]];
    CONST robtarget Target_65_2:=[[-119.958,-120.121,103.016],[0,-0.707106781,0.707106781,0],[-2,-1,-1,0],[9E+09,9E+09,9E+09,9E+09,9E+09,9E+09]];
    CONST robtarget Target_70_2:=[[-119.958,-120.121,53.016],[0,-0.707106781,0.707106781,0],[-2,-1,0,0],[9E+09,9E+09,9E+09,9E+09,9E+09,9E+09]];
    CONST robtarget Target_75_2:=[[-119.992,-200.079,103.016],[0,-0.707106781,0.707106781,0],[-2,-1,-1,0],[9E+09,9E+09,9E+09,9E+09,9E+09,9E+09]];
    CONST robtarget Target_80_2:=[[-119.992,-200.079,53.016],[0,-0.707106781,0.707106781,0],[-2,-1,0,0],[9E+09,9E+09,9E+09,9E+09,9E+09,9E+09]];
    CONST robtarget Target_85_2:=[[-200.003,-40.005,103.016],[0,-0.707106781,0.707106781,0],[-2,-1,-1,0],[9E+09,9E+09,9E+09,9E+09,9E+09,9E+09]];
    CONST robtarget Target_90_2:=[[-200.003,-40.005,53.016],[0,-0.707106781,0.707106781,0],[-2,-1,-1,0],[9E+09,9E+09,9E+09,9E+09,9E+09,9E+09]];
    CONST robtarget Target_95_2:=[[-200.003,-120.004,103.016],[0,-0.707106781,0.707106781,0],[-2,-1,-1,0],[9E+09,9E+09,9E+09,9E+09,9E+09,9E+09]];
    CONST robtarget Target_100_2:=[[-200.003,-120.004,53.016],[0,-0.707106781,0.707106781,0],[-2,-1,-1,0],[9E+09,9E+09,9E+09,9E+09,9E+09,9E+09]];
    CONST robtarget Target_105_2:=[[-200.003,-200.005,103.016],[0,-0.707106781,0.707106781,0],[-2,-1,-1,0],[9E+09,9E+09,9E+09,9E+09,9E+09,9E+09]];
    CONST robtarget Target_110_2:=[[-200.003,-200.005,53.016],[0,-0.707106781,0.707106781,0],[-2,-1,-1,0],[9E+09,9E+09,9E+09,9E+09,9E+09,9E+09]];
    CONST robtarget Target_112:=[[-104.999986788,268.411364612,-142.18870844],[0.000000009,-0.000000017,-0.707106759,0.707106803],[-1,0,-1,0],[9E+09,9E+09,9E+09,9E+09,9E+09,9E+09]];
    CONST robtarget Target_115:=[[-105,70,-267],[0,0,-0.707106781,0.707106781],[-1,0,-2,0],[9E+09,9E+09,9E+09,9E+09,9E+09,9E+09]];
    CONST robtarget Target_120:=[[-105,5,-267],[0,0,-0.707106781,0.707106781],[0,1,-2,0],[9E+09,9E+09,9E+09,9E+09,9E+09,9E+09]];

    PROC main()
        SetDO Attach_pieza_acople,0;
        SetDO Detach_pieza_acople,1;
        SetDO Attach_pieza_desacople,0;
        SetDO Detach_pieza_desacople,1;
        SetDO Start_torno_1,0;
        SetDO Start_torno_2,0;
        SetDO Start_giro,0;
        SetDO Tool_acople_activa,0;
        SetDO Tool_desacople_activa,0;
        WHILE TRUE DO
            restartObjetivos;
            Configurar_inicial;
            !Add your code here
            Home2_a_home1;
            WaitTime 1;
            IF SinMaquinar1 = 1 THEN
                Agarrar_pieza_1;
            ELSEIF SinMaquinar2 = 1 THEN
                Agarrar_pieza_2;
            ELSEIF SinMaquinar3 = 1 THEN
                Agarrar_pieza_3;
            ELSEIF SinMaquinar4 = 1 THEN
                Agarrar_pieza_4;
            ELSEIF SinMaquinar5 = 1 THEN
                Agarrar_pieza_5;
            ELSEIF SinMaquinar6 = 1 THEN
                Agarrar_pieza_6;
            ELSEIF SinMaquinar7 = 1 THEN
                Agarrar_pieza_7;
            ELSEIF SinMaquinar8 = 1 THEN
                Agarrar_pieza_8;
            ELSEIF SinMaquinar9 = 1 THEN
                Agarrar_pieza_9;
            ELSE
                continue := FALSE;
            ENDIF

            restartObjetivos;
            IF continue = FALSE THEN
                IF Torno_2_has_mounted = 1 THEN
                    Ir_a_torno_2;
                ENDIF

                IF Tool_desacople_activa = 1 THEN
                    IF Maquinada9 = 0 THEN
                        Terminar_pieza_9;
                    ELSEIF Maquinada8 = 0 THEN
                        Terminar_pieza_8;
                    ELSEIF Maquinada7 = 0 THEN
                        Terminar_pieza_7;
                    ELSEIF Maquinada6 = 0 THEN
                        Terminar_pieza_6;
                    ELSEIF Maquinada5 = 0 THEN
                        Terminar_pieza_5;
                    ELSEIF Maquinada4 = 0 THEN
                        Terminar_pieza_4;
                    ELSEIF Maquinada3 = 0 THEN
                        Terminar_pieza_3;
                    ELSEIF Maquinada2 = 0 THEN
                        Terminar_pieza_2;
                    ELSEIF Maquinada1 = 0 THEN
                        Terminar_pieza_1;
                    ENDIF
                ENDIF
            ELSE
                Ir_a_torno_1;
                IF Tool_desacople_activa = 1 THEN
                    Girar_pieza;
                    Ir_a_torno_2;
                    IF Tool_desacople_activa = 1 THEN
                        IF Maquinada9 = 0 THEN
                            Terminar_pieza_9;
                        ELSEIF Maquinada8 = 0 THEN
                            Terminar_pieza_8;
                        ELSEIF Maquinada7 = 0 THEN
                            Terminar_pieza_7;
                        ELSEIF Maquinada6 = 0 THEN
                            Terminar_pieza_6;
                        ELSEIF Maquinada5 = 0 THEN
                            Terminar_pieza_5;
                        ELSEIF Maquinada4 = 0 THEN
                            Terminar_pieza_4;
                        ELSEIF Maquinada3 = 0 THEN
                            Terminar_pieza_3;
                        ELSEIF Maquinada2 = 0 THEN
                            Terminar_pieza_2;
                        ELSEIF Maquinada1 = 0 THEN
                            Terminar_pieza_1;
                        ENDIF
                    ENDIF
                ENDIF
            ENDIF

        ENDWHILE


    ENDPROC
    PROC Configurar_inicial()
        IF SinMaquinar1 = 1 THEN
            SetDO Pieza_1_objetivo,1;
        ELSEIF SinMaquinar2 = 1 THEN
            SetDO Pieza_2_objetivo,1;
        ELSEIF SinMaquinar3 = 1 THEN
            SetDO Pieza_3_objetivo,1;
        ELSEIF SinMaquinar4 = 1 THEN
            SetDO Pieza_4_objetivo,1;
        ELSEIF SinMaquinar5 = 1 THEN
            SetDO Pieza_5_objetivo,1;
        ELSEIF SinMaquinar6 = 1 THEN
            SetDO Pieza_6_objetivo,1;
        ELSEIF SinMaquinar7 = 1 THEN
            SetDO Pieza_7_objetivo,1;
        ELSEIF SinMaquinar8 = 1 THEN
            SetDO Pieza_8_objetivo,1;
        ELSEIF SinMaquinar9 = 1 THEN
            SetDO Pieza_9_objetivo,1;
        ELSE
            continue := FALSE;
        ENDIF

        IF Maquinada9 = 0 THEN
            contador_maquinadas := 9;
        ELSEIF Maquinada8 = 0 THEN
            contador_maquinadas := 8;
        ELSEIF Maquinada7 = 0 THEN
            contador_maquinadas := 7;
        ELSEIF Maquinada6 = 0 THEN
            contador_maquinadas := 6;
        ELSEIF Maquinada5 = 0 THEN
            contador_maquinadas := 5;
        ELSEIF Maquinada4 = 0 THEN
            contador_maquinadas := 4;
        ELSEIF Maquinada3 = 0 THEN
            contador_maquinadas := 3;
        ELSEIF Maquinada2 = 0 THEN
            contador_maquinadas := 2;
        ELSEIF Maquinada1 = 0 THEN
            contador_maquinadas := 1;
        ELSE
            continue := FALSE;
        ENDIF
    ENDPROC

    PROC definirObjetivo()
        IF contador_sin_maquinar = 1 THEN
            SetDO Pieza_1_objetivo,1;
        ELSEIF contador_sin_maquinar = 2 THEN
            SetDO Pieza_2_objetivo,1;
        ELSEIF contador_sin_maquinar = 3 THEN
            SetDO Pieza_3_objetivo,1;
        ELSEIF contador_sin_maquinar = 4 THEN
            SetDO Pieza_4_objetivo,1;
        ELSEIF contador_sin_maquinar = 5 THEN
            SetDO Pieza_5_objetivo,1;
        ELSEIF contador_sin_maquinar = 6 THEN
            SetDO Pieza_6_objetivo,1;
        ELSEIF contador_sin_maquinar = 7 THEN
            SetDO Pieza_7_objetivo,1;
        ELSEIF contador_sin_maquinar = 8 THEN
            SetDO Pieza_8_objetivo,1;
        ELSEIF contador_sin_maquinar = 9 THEN
            SetDO Pieza_9_objetivo,1;
        ENDIF
    ENDPROC

    PROC restartObjetivos()
        SetDO Pieza_1_objetivo,0;
        SetDO Pieza_2_objetivo,0;
        SetDO Pieza_3_objetivo,0;
        SetDO Pieza_4_objetivo,0;
        SetDO Pieza_5_objetivo,0;
        SetDO Pieza_6_objetivo,0;
        SetDO Pieza_7_objetivo,0;
        SetDO Pieza_8_objetivo,0;
        SetDO Pieza_9_objetivo,0;
    ENDPROC
    PROC Ir_a_torno_1()
        MoveJ Target_0,v400,z100,Refrigerator\WObj:=Workobject_3;
        MoveJ Target_3,v400,z100,Tool_desacople\WObj:=Workobject_3;
        MoveJ Target_5,v400,z5,Tool_desacople\WObj:=Workobject_3;
        IF Torno_1_has_mounted = 1 THEN
            Quitar_pieza_1;
        ENDIF
        IF Tool_acople_activa = 1 THEN
            Refrigerar_1;
            Colocar_pieza_1;
        ENDIF

        Volver_1;
    ENDPROC
    PROC Quitar_pieza_1()
        MoveL Target_10,v50,z5,Tool_desacople\WObj:=Workobject_3;
        WaitTime 1;
        SetDO Attach_pieza_desacople,1;
        SetDO Detach_pieza_desacople,0;
        SetDO Tool_desacople_activa,1;
        SetDO Start_torno_1,0;
        MoveL Target_5,v50,z5,Tool_desacople\WObj:=Workobject_3;
    ENDPROC
    PROC Refrigerar_1()
        MoveJ Target_5,v400,z100,Tool_desacople\WObj:=Workobject_3;
        MoveJ Target_5,v400,z100,Refrigerator\WObj:=Workobject_3;
        MoveL Target_10,v50,z5,Refrigerator\WObj:=Workobject_3;
        MoveL Target_5,v50,z5,Refrigerator\WObj:=Workobject_3;
        MoveL Target_10,v50,z5,Refrigerator\WObj:=Workobject_3;
        MoveL Target_5,v50,z5,Refrigerator\WObj:=Workobject_3;
    ENDPROC
    PROC Colocar_pieza_1()
        MoveJ Target_5,v400,z100,Tool_acople\WObj:=Workobject_3;
        MoveL Target_10,v50,z5,Tool_acople\WObj:=Workobject_3;
        WaitTime 1;
        SetDO Attach_pieza_acople,0;
        SetDO Detach_pieza_acople,1;
        SetDO Tool_acople_activa,0;
        SetDO Start_torno_1,1;
        MoveL Target_5,v50,z5,Tool_acople\WObj:=Workobject_3;
    ENDPROC
    PROC Volver_1()
        MoveJ Target_5,v400,z100,Tool_desacople\WObj:=Workobject_3;
        MoveJ Target_3,v400,z100,Tool_desacople\WObj:=Workobject_3;
        MoveJ Target_0,v400,z100,Refrigerator\WObj:=Workobject_3;
    ENDPROC
    PROC Quitar_pieza_2()
        MoveL Target_10_2,v50,z5,Tool_desacople\WObj:=Workobject_4;
        WaitTime 1;
        SetDO Attach_pieza_desacople,1;
        SetDO Detach_pieza_desacople,0;
        SetDO Tool_desacople_activa,1;
        SetDO Start_torno_2,0;
        MoveL Target_5_2,v50,z5,Tool_desacople\WObj:=Workobject_4;
    ENDPROC
    PROC Refrigerar_2()
        MoveJ Target_5_2,v400,z100,Tool_desacople\WObj:=Workobject_4;
        MoveJ Target_5_2,v400,z100,Refrigerator\WObj:=Workobject_4;
        MoveL Target_10_2,v50,z5,Refrigerator\WObj:=Workobject_4;
        MoveL Target_5_2,v50,z5,Refrigerator\WObj:=Workobject_4;
        MoveL Target_10_2,v50,z5,Refrigerator\WObj:=Workobject_4;
        MoveL Target_5_2,v50,z5,Refrigerator\WObj:=Workobject_4;
    ENDPROC
    PROC Colocar_pieza_2()
        MoveJ Target_5_2,v400,z100,Tool_acople\WObj:=Workobject_4;
        MoveL Target_10_2,v50,z5,Tool_acople\WObj:=Workobject_4;
        WaitTime 1;
        SetDO Attach_pieza_acople,0;
        SetDO Detach_pieza_acople,1;
        SetDO Tool_acople_activa,0;
        SetDO Start_torno_2,1;
        MoveL Target_5_2,v50,z5,Tool_acople\WObj:=Workobject_4;
    ENDPROC
    PROC Ir_a_torno_2()
        MoveJ Target_0_3,v400,z100,Refrigerator\WObj:=Workobject_2;
        MoveJ Target_3_2,v400,z100,Tool_desacople\WObj:=Workobject_4;
        MoveJ Target_5_2,v400,z100,Tool_desacople\WObj:=Workobject_4;
        IF Torno_2_has_mounted = 1 THEN
            Quitar_pieza_2;
        ENDIF

        IF Tool_acople_activa = 1 THEN
            Refrigerar_2;
            Colocar_pieza_2;
        ENDIF

        Volver_2;
    ENDPROC
    PROC Volver_2()
        MoveJ Target_5_2,v400,z100,Tool_desacople\WObj:=Workobject_4;
        MoveJ Target_3_2,v400,z100,Tool_desacople\WObj:=Workobject_4;
        MoveJ Target_0_3,v400,z100,Refrigerator\WObj:=Workobject_2;
    ENDPROC
    PROC Agarrar_pieza_1()
        MoveJ Target_25,v400,z100,Tool_acople\WObj:=Workobject_1;
        MoveL Target_30,v50,z5,Tool_acople\WObj:=Workobject_1;
        WaitTime 1;
        SetDO Attach_pieza_acople,1;
        SetDO Detach_pieza_acople,0;
        SetDO Tool_acople_activa,1;
        MoveL Target_25,v50,z5,Tool_acople\WObj:=Workobject_1;
        MoveJ Target_0,v400,z100,Refrigerator\WObj:=Workobject_3;
    ENDPROC
    PROC Agarrar_pieza_2()
        MoveJ Target_35,v400,z100,Tool_acople\WObj:=Workobject_1;
        MoveL Target_40,v50,z5,Tool_acople\WObj:=Workobject_1;
        WaitTime 1;
        SetDO Attach_pieza_acople,1;
        SetDO Detach_pieza_acople,0;
        SetDO Tool_acople_activa,1;
        MoveL Target_35,v50,z5,Tool_acople\WObj:=Workobject_1;
        MoveJ Target_0,v400,z100,Refrigerator\WObj:=Workobject_3;
    ENDPROC
    PROC Agarrar_pieza_3()
        MoveJ Target_45,v400,z100,Tool_acople\WObj:=Workobject_1;
        MoveL Target_50,v50,z5,Tool_acople\WObj:=Workobject_1;
        WaitTime 1;
        SetDO Attach_pieza_acople,1;
        SetDO Detach_pieza_acople,0;
        SetDO Tool_acople_activa,1;
        MoveL Target_45,v50,z5,Tool_acople\WObj:=Workobject_1;
        MoveJ Target_0,v400,z100,Refrigerator\WObj:=Workobject_3;
    ENDPROC
    PROC Agarrar_pieza_4()
        MoveJ Target_55,v400,z100,Tool_acople\WObj:=Workobject_1;
        MoveL Target_60,v50,z5,Tool_acople\WObj:=Workobject_1;
        WaitTime 1;
        SetDO Attach_pieza_acople,1;
        SetDO Detach_pieza_acople,0;
        SetDO Tool_acople_activa,1;
        MoveL Target_55,v50,z5,Tool_acople\WObj:=Workobject_1;
        MoveJ Target_0,v400,z100,Refrigerator\WObj:=Workobject_3;
    ENDPROC
    PROC Agarrar_pieza_5()
        MoveJ Target_65,v400,z100,Tool_acople\WObj:=Workobject_1;
        MoveL Target_70,v50,z5,Tool_acople\WObj:=Workobject_1;
        WaitTime 1;
        SetDO Attach_pieza_acople,1;
        SetDO Detach_pieza_acople,0;
        SetDO Tool_acople_activa,1;
        MoveL Target_65,v50,z5,Tool_acople\WObj:=Workobject_1;
        MoveJ Target_0,v400,z100,Refrigerator\WObj:=Workobject_3;
    ENDPROC
    PROC Agarrar_pieza_6()
        MoveJ Target_75,v400,z100,Tool_acople\WObj:=Workobject_1;
        MoveL Target_80,v50,z5,Tool_acople\WObj:=Workobject_1;
        WaitTime 1;
        SetDO Attach_pieza_acople,1;
        SetDO Detach_pieza_acople,0;
        SetDO Tool_acople_activa,1;
        MoveL Target_75,v50,z5,Tool_acople\WObj:=Workobject_1;
        MoveJ Target_0,v400,z100,Refrigerator\WObj:=Workobject_3;
    ENDPROC
    PROC Agarrar_pieza_7()
        MoveJ Target_85,v400,z100,Tool_acople\WObj:=Workobject_1;
        MoveL Target_90,v50,z5,Tool_acople\WObj:=Workobject_1;
        WaitTime 1;
        SetDO Attach_pieza_acople,1;
        SetDO Detach_pieza_acople,0;
        SetDO Tool_acople_activa,1;
        MoveL Target_85,v50,z5,Tool_acople\WObj:=Workobject_1;
        MoveJ Target_0,v400,z100,Refrigerator\WObj:=Workobject_3;
    ENDPROC
    PROC Agarrar_pieza_8()
        MoveJ Target_95,v400,z100,Tool_acople\WObj:=Workobject_1;
        MoveL Target_100,v50,z5,Tool_acople\WObj:=Workobject_1;
        WaitTime 1;
        SetDO Attach_pieza_acople,1;
        SetDO Detach_pieza_acople,0;
        SetDO Tool_acople_activa,1;
        MoveL Target_95,v50,z5,Tool_acople\WObj:=Workobject_1;
        MoveJ Target_0,v400,z100,Refrigerator\WObj:=Workobject_3;
    ENDPROC
    PROC Agarrar_pieza_9()
        MoveJ Target_105,v400,z100,Tool_acople\WObj:=Workobject_1;
        MoveL Target_110,v50,z5,Tool_acople\WObj:=Workobject_1;
        WaitTime 1;
        SetDO Attach_pieza_acople,1;
        SetDO Detach_pieza_acople,0;
        SetDO Tool_acople_activa,1;
        MoveL Target_105,v50,z5,Tool_acople\WObj:=Workobject_1;
        MoveJ Target_0_4,v400,z100,Refrigerator\WObj:=Workobject_3;
    ENDPROC
    PROC Terminar_pieza_1()
        MoveJ Target_25_2,v400,z100,Tool_desacople\WObj:=Workobject_2;
        MoveL Target_30_2,v50,z5,Tool_desacople\WObj:=Workobject_2;
        WaitTime 1;
        SetDO Attach_pieza_desacople,0;
        SetDO Detach_pieza_desacople,1;
        SetDO Tool_desacople_activa,0;
        MoveL Target_25_2,v50,z5,Tool_desacople\WObj:=Workobject_2;
        MoveJ Target_0_3,v400,z100,Refrigerator\WObj:=Workobject_2;
    ENDPROC
    PROC Terminar_pieza_2()
        MoveJ Target_35_2,v400,z100,Tool_desacople\WObj:=Workobject_2;
        MoveL Target_40_2,v50,z5,Tool_desacople\WObj:=Workobject_2;
        WaitTime 1;
        SetDO Attach_pieza_desacople,0;
        SetDO Detach_pieza_desacople,1;
        SetDO Tool_desacople_activa,0;
        MoveL Target_35_2,v50,z5,Tool_desacople\WObj:=Workobject_2;
        MoveJ Target_0_3,v400,z100,Refrigerator\WObj:=Workobject_2;
    ENDPROC
    PROC Terminar_pieza_3()
        MoveJ Target_45_2,v400,z100,Tool_desacople\WObj:=Workobject_2;
        MoveL Target_50_2,v50,z5,Tool_desacople\WObj:=Workobject_2;
        WaitTime 1;
        SetDO Attach_pieza_desacople,0;
        SetDO Detach_pieza_desacople,1;
        SetDO Tool_desacople_activa,0;
        MoveL Target_45_2,v50,z5,Tool_desacople\WObj:=Workobject_2;
        MoveJ Target_0_3,v400,z100,Refrigerator\WObj:=Workobject_2;
    ENDPROC
    PROC Terminar_pieza_4()
        MoveJ Target_55_2,v400,z100,Tool_desacople\WObj:=Workobject_2;
        MoveL Target_60_2,v50,z5,Tool_desacople\WObj:=Workobject_2;
        WaitTime 1;
        SetDO Attach_pieza_desacople,0;
        SetDO Detach_pieza_desacople,1;
        SetDO Tool_desacople_activa,0;
        MoveL Target_55_2,v50,z5,Tool_desacople\WObj:=Workobject_2;
        MoveJ Target_0_3,v400,z100,Refrigerator\WObj:=Workobject_2;
    ENDPROC
    PROC Terminar_pieza_5()
        MoveJ Target_65_2,v400,z100,Tool_desacople\WObj:=Workobject_2;
        MoveL Target_70_2,v50,z5,Tool_desacople\WObj:=Workobject_2;
        WaitTime 1;
        SetDO Attach_pieza_desacople,0;
        SetDO Detach_pieza_desacople,1;
        SetDO Tool_desacople_activa,0;
        MoveL Target_65_2,v50,z5,Tool_desacople\WObj:=Workobject_2;
        MoveJ Target_0_3,v400,z100,Refrigerator\WObj:=Workobject_2;
    ENDPROC
    PROC Terminar_pieza_6()
        MoveJ Target_75_2,v400,z100,Tool_desacople\WObj:=Workobject_2;
        MoveL Target_80_2,v50,z5,Tool_desacople\WObj:=Workobject_2;
        WaitTime 1;
        SetDO Attach_pieza_desacople,0;
        SetDO Detach_pieza_desacople,1;
        SetDO Tool_desacople_activa,0;
        MoveL Target_75_2,v50,z5,Tool_desacople\WObj:=Workobject_2;
        MoveJ Target_0_3,v400,z100,Refrigerator\WObj:=Workobject_2;
    ENDPROC
    PROC Terminar_pieza_7()
        MoveJ Target_85_2,v400,z100,Tool_desacople\WObj:=Workobject_2;
        MoveL Target_90_2,v50,z5,Tool_desacople\WObj:=Workobject_2;
        WaitTime 1;
        SetDO Attach_pieza_desacople,0;
        SetDO Detach_pieza_desacople,1;
        SetDO Tool_desacople_activa,0;
        MoveL Target_85_2,v50,z5,Tool_desacople\WObj:=Workobject_2;
        MoveJ Target_0_3,v400,z100,Refrigerator\WObj:=Workobject_2;
    ENDPROC
    PROC Terminar_pieza_8()
        MoveJ Target_95_2,v400,z100,Tool_desacople\WObj:=Workobject_2;
        MoveL Target_100_2,v50,z5,Tool_desacople\WObj:=Workobject_2;
        WaitTime 1;
        SetDO Attach_pieza_desacople,0;
        SetDO Detach_pieza_desacople,1;
        SetDO Tool_desacople_activa,0;
        MoveL Target_95_2,v50,z5,Tool_desacople\WObj:=Workobject_2;
        MoveJ Target_0_3,v400,z100,Refrigerator\WObj:=Workobject_2;
    ENDPROC
    PROC Terminar_pieza_9()
        MoveJ Target_105_2,v400,z100,Tool_desacople\WObj:=Workobject_2;
        MoveL Target_110_2,v50,z5,Tool_desacople\WObj:=Workobject_2;
        WaitTime 1;
        SetDO Attach_pieza_desacople,0;
        SetDO Detach_pieza_desacople,1;
        SetDO Tool_desacople_activa,0;
        MoveL Target_105_2,v50,z5,Tool_desacople\WObj:=Workobject_2;
        MoveJ Target_0_3,v400,z100,Refrigerator\WObj:=Workobject_2;
    ENDPROC
    PROC Home2_a_home1()
        MoveJ Target_0,v400,z100,Refrigerator\WObj:=Workobject_3;
    ENDPROC
    PROC Girar_pieza()
        MoveJ Target_112,v400,z100,Tool_desacople\WObj:=Workobject_1;
        MoveJ Target_115,v400,z100,Tool_desacople\WObj:=Workobject_1;
        MoveL Target_120,v50,z5,Tool_desacople\WObj:=Workobject_1;
        WaitTime 1;
        SetDO Attach_pieza_desacople,0;
        SetDO Detach_pieza_desacople,1;
        SetDO Tool_desacople_activa,0;
        SetDO Start_giro,1;
        MoveL Target_115,v50,z5,Tool_desacople\WObj:=Workobject_1;
        MoveJ Target_115,v400,z100,Tool_acople\WObj:=Workobject_1;
        WaitTime 3;
        MoveL Target_120,v50,z5,Tool_acople\WObj:=Workobject_1;
        WaitTime 1;
        SetDO Attach_pieza_acople,1;
        SetDO Detach_pieza_acople,0;
        SetDO Tool_acople_activa,1;
        SetDO Start_giro,0;
        MoveL Target_115,v50,z5,Tool_acople\WObj:=Workobject_1;
        MoveJ Target_112,v400,z100,Tool_desacople\WObj:=Workobject_1;
        MoveJ Target_0,v400,z100,Refrigerator\WObj:=Workobject_3;
    ENDPROC
ENDMODULE

--- Backups/Controller8/SYSPAR/EIO.cfg ---
EIO:CFG_1.0:6:1::
#
EIO_SIGNAL:

      -Name "SinMaquinar1" -SignalType "DI"

      -Name "SinMaquinar2" -SignalType "DI"

      -Name "SinMaquinar3" -SignalType "DI"

      -Name "SinMaquinar4" -SignalType "DI"

      -Name "SinMaquinar5" -SignalType "DI"

      -Name "SinMaquinar6" -SignalType "DI"

      -Name "SinMaquinar7" -SignalType "DI"

      -Name "SinMaquinar8" -SignalType "DI"

      -Name "SinMaquinar9" -SignalType "DI"

      -Name "Maquinada1" -SignalType "DI"

      -Name "Maquinada2" -SignalType "DI"

      -Name "Maquinada3" -SignalType "DI"

      -Name "Maquinada4" -SignalType "DI"

      -Name "Maquinada5" -SignalType "DI"

      -Name "Maquinada6" -SignalType "DI"

      -Name "Maquinada7" -SignalType "DI"

      -Name "Maquinada8" -SignalType "DI"

      -Name "Maquinada9" -SignalType "DI"

      -Name "Torno_1_finished" -SignalType "DI"

      -Name "Torno_2_finished" -SignalType "DI"

      -Name "Torno_1_has_mounted" -SignalType "DI"

      -Name "Torno_2_has_mounted" -SignalType "DI"

      -Name "Rotated" -SignalType "DI"

      -Name "Tool_acople_activa" -SignalType "DO"

      -Name "Tool_desacople_activa" -SignalType "DO"

      -Name "Start_torno_1" -SignalType "DO"

      -Name "Start_torno_2" -SignalType "DO"

      -Name "Start_giro" -SignalType "DO"

      -Name "Attach_pieza_acople" -SignalType "DO"

      -Name "Detach_pieza_acople" -SignalType "DO"

      -Name "Pieza_1_objetivo" -SignalType "DO"

      -Name "Pieza_2_objetivo" -SignalType "DO"

      -Name "Pieza_3_objetivo" -SignalType "DO"

      -Name "Pieza_4_objetivo" -SignalType "DO"

      -Name "Pieza_5_objetivo" -SignalType "DO"

      -Name "Pieza_6_objetivo" -SignalType "DO"

      -Name "Pieza_7_objetivo" -SignalType "DO"

      -Name "Pieza_8_objetivo" -SignalType "DO"

      -Name "Pieza_9_objetivo" -SignalType "DO"

      -Name "Attach_pieza_desacople" -SignalType "DO"

      -Name "Detach_pieza_desacople" -SignalType "DO"
